(* Schneider Machine Expert - Basic project P1-Part1A, file version 1.6.0.0 *)
(* ProjectInformations: Name=New project *)

HARDWARE
  Cpu 0: TM221M16R/G
  EthernetConfiguration: NetworkName=M221, IpAllocationMode=FixedAddress, IpAddress=0.0.0.0, SubnetMask=0.0.0.0
  SerialLineConfiguration: Baud=Baud19200, Parity=ParityEven, DataBits=DataBits8, StopBits=StopBits1, PhysicalMedium=PhysicalMediumRs485, TransmissionMode=TransmissionModeModbusRtu, SlaveId=1, Addressing=SlaveAddressing
  MastTask: UsePeriodScanMode=false, PeriodScan=100
  FastTask: Period=255
  CpuBehavior: StartingMode=StartAsPreviousState, AutoSaveRamOnEeprom=true, WatchdogPeriod=250

SYMBOLS  (address, symbol, comment, settings)
  %MW0      CURRENT_PRESSURE
  %KW0      PRESSURE_CHECKPOINT  [Value=500]
  %KW1      PRESSURE_CHECKPOINT_UNREACHABLE  [Value=1001]
  %I0.0     INPUT_0
  %I0.1     INPUT_1
  %Q0.0     OUTPUT_0
  %Q0.1     OUTPUT_1

POU I/O Control  (* I/O and Timer Control *)
  (* SectionNumber=1 *)

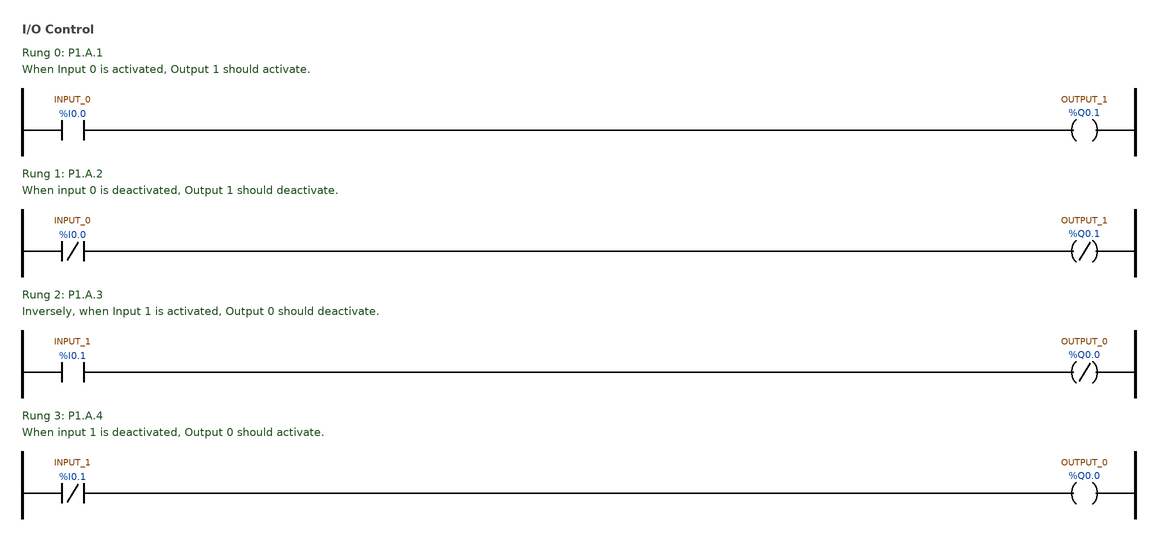

// Rung 0: P1.A.1
// When Input 0 is activated, Output 1 should activate.
  LD %I0.0                (* INPUT_0 *)
  ST %Q0.1                (* OUTPUT_1 *)
  // as ST:
  //   OUTPUT_1 := INPUT_0;

// Rung 1: P1.A.2
// When input 0 is deactivated, Output 1 should deactivate.
  LDN %I0.0               (* INPUT_0 *)
  STN %Q0.1               (* OUTPUT_1 *)
  // as ST:
  //   OUTPUT_1 := NOT (NOT INPUT_0);

// Rung 2: P1.A.3
// Inversely, when Input 1 is activated, Output 0 should deactivate.
  LD %I0.1                (* INPUT_1 *)
  STN %Q0.0               (* OUTPUT_0 *)
  // as ST:
  //   OUTPUT_0 := NOT INPUT_1;

// Rung 3: P1.A.4
// When input 1 is deactivated, Output 0 should activate.
  LDN %I0.1               (* INPUT_1 *)
  ST %Q0.0                (* OUTPUT_0 *)
  // as ST:
  //   OUTPUT_0 := NOT INPUT_1;
